(* IEC 61131-3 sources: AcpTrakStarwheel/TrkBufLib, 10 files *)

(* ---- Types.typ ---- *)
(*Buffer Base Type*)

TYPE
	tbAsyncShuttleBufferType : 	STRUCT  (*Asynchronous Buffer data*)
		ReadIdx : USINT; (*Starting index of the ring buffer*)
		WriteIdx : USINT; (*Ending index of the ring buffer*)
		Shuttles : ARRAY[0..tbMAX_BUF_IDX]OF McAxisType; (*Shuttles in the ring buffer*)
	END_STRUCT;
END_TYPE

(*Routed Move Velcity from Trigger Buffer*)

TYPE
	tbRtdMvVelTrgBufferParType : 	STRUCT  (*Parameters*)
		Position : LREAL; (*Position to send shuttle to*)
		RouteVelocity : REAL; (*Velocity of the shuttle before reaching the target position*)
		Velocity : REAL; (*Velocity of the shuttle after reaching the target position*)
		Acceleration : REAL; (*Acceleration of shuttle*)
		Deceleration : REAL; (*Deceleration of shuttle*)
		AdvancedParameters : McAcpTrakAdvRouteParType; (*Advanced move parameters*)
	END_STRUCT;
	tbRtdMvVelTrgBufferInternalType : 	STRUCT  (*Internal Data*)
		State : tbRtdTrgBufferStateEnum; (*State of execution*)
		TrgPointEnable : MC_BR_TrgPointEnable_AcpTrak; (*Enable process point*)
		TrgPointGetInfo : MC_BR_TrgPointGetInfo_AcpTrak; (*Get process point information*)
		RoutedMoveVel : MC_BR_RoutedMoveVel_AcpTrak; (*Move shuttle*)
		Status : DINT; (*Status*)
	END_STRUCT;
	tbRtdTrgBufferStateEnum :
		( (*State of execution for routed move from trigger*)
		tbRTD_TRG_BUF_STATE_IDLE, (*Idle state*)
		tbRTD_TRG_BUF_STATE_ENABLE_TRIG, (*Enable the process point*)
		tbRTD_TRG_BUF_STATE_GET_INFO, (*Get information from the start process point*)
		tbRTD_TRG_BUF_STATE_MOVE, (*Move shuttle*)
		tbRTD_TRG_BUF_STATE_RESET_FB, (*Reset function blocks*)
		tbRTD_TRG_BUF_STATE_NOT_BUSY, (*Wait for function blocks to report not busy*)
		tbRTD_TRG_BUF_STATE_ERROR (*An error occurred*)
		);
END_TYPE

(*Elastic Move Absolute from Position Buffer*)

TYPE
	tbElaMvAbsPosBufferParType : 	STRUCT  (*Parameters*)
		ArrivalPosition : LREAL; (*Position to wait for shuttles to arrive to*)
		DestinationPosition : LREAL; (*Position to send shuttles to*)
		DestinationVelocity : REAL; (*Velocity to move to destination*)
		DestinationAcceleration : REAL; (*Acceleration to move to destination*)
		DestinationDeceleration : REAL; (*Deceleration to move to destination*)
	END_STRUCT;
	tbElaMvAbsPosBufferInternalType : 	STRUCT  (*Internal Data*)
		State : tbElaPosBufferStateEnum; (*State of execution*)
		ShReadInfo : MC_BR_ShReadInfo_AcpTrak; (*Read shuttle info*)
		ElasticMoveAbs : MC_BR_ElasticMoveAbs_AcpTrak; (*Elastic move absolute*)
		Axis : McAxisType; (*Axis to control*)
		Status : DINT; (*Status*)
	END_STRUCT;
	tbElaPosBufferStateEnum :
		( (*State of execution*)
		tbELA_POS_BUF_STATE_IDLE, (*Idle state*)
		tbELA_POS_BUF_STATE_WAIT, (*Wait for a shuttle to be available*)
		tbELA_POS_BUF_STATE_POS, (*Wait for shuttle to reach the specified position on the sector*)
		tbELA_POS_BUF_STATE_MOVE, (*Move the shuttle to its position*)
		tbELA_POS_BUF_STATE_RESET_FB, (*Reset function blocks*)
		tbELA_POS_BUF_STATE_NOT_BUSY, (*Wait for function blocks to report not busy*)
		tbELA_POS_BUF_STATE_ERROR (*An error occurred*)
		);
END_TYPE

(* ---- BufferAddSh.st ---- *)
FUNCTION tbBufferAddSh

    IF ((Buffer.WriteIdx + 1) MOD (tbMAX_BUF_IDX + 1)) = Buffer.ReadIdx THEN
       tbBufferAddSh := tbERR_MAX_BUF_IDX;
    ELSE
        //Add the shuttle to the buffer
        brsmemcpy(ADR(Buffer.Shuttles[Buffer.WriteIdx]), ADR(Shuttle), SIZEOF(Buffer.Shuttles[Buffer.WriteIdx]));
        Buffer.WriteIdx := (Buffer.WriteIdx + 1) MOD (tbMAX_BUF_IDX + 1);
        tbBufferAddSh := ERR_OK;
    END_IF
    RETURN;

END_FUNCTION

(* ---- BufferGetFirst.st ---- *)
FUNCTION tbBufferGetFirst

    IF tbBufferShAvailable(ADR(Buffer)) THEN
        brsmemcpy(ADR(Shuttle), ADR(Buffer.Shuttles[Buffer.ReadIdx]), SIZEOF(Shuttle));
        tbBufferGetFirst := ERR_OK;
    ELSE
        tbBufferGetFirst := tbERR_NO_SH_IN_BUFFER;
    END_IF
    RETURN;

END_FUNCTION

(* ---- BufferRemoveFirst.st ---- *)
FUNCTION tbBufferRemoveFirst

    IF tbBufferShAvailable(ADR(Buffer)) THEN
        Buffer.ReadIdx := (Buffer.ReadIdx + 1) MOD (tbMAX_BUF_IDX + 1);
        tbBufferRemoveFirst := ERR_OK;
    ELSE
        tbBufferRemoveFirst := tbERR_NO_SH_IN_BUFFER;
    END_IF
    RETURN;

END_FUNCTION

(* ---- BufferShAvailable.st ---- *)
FUNCTION tbBufferShAvailable

    tbBufferShAvailable := Buffer.ReadIdx <> Buffer.WriteIdx;
    RETURN;

END_FUNCTION

(* ---- ShInBuffer.st ---- *)
FUNCTION tbShInBuffer

    i := Buffer.ReadIdx;
    WHILE i <> Buffer.WriteIdx DO
        IF brsmemcmp(ADR(Buffer.Shuttles[i]), ADR(Shuttle), SIZEOF(Buffer.Shuttles[i])) = 0 THEN
            tbShInBuffer := 1;
            RETURN;
        END_IF
        i := (i + 1) MOD (tbMAX_BUF_IDX + 1);
    END_WHILE
    tbShInBuffer := 0;
    RETURN;

END_FUNCTION

(* ---- ElasticMoveAbsPosBuffer.st ---- *)
FUNCTION_BLOCK tbElasticMoveAbsPosBuffer

    CASE Internal.State OF

        tbELA_POS_BUF_STATE_IDLE:

            IF Enable THEN
                Busy := 1;
                Active := 1;
                Internal.ShReadInfo.Axis := ADR(Internal.Axis);
                Internal.ElasticMoveAbs.Axis := ADR(Internal.Axis);
                Internal.State := tbELA_POS_BUF_STATE_WAIT;
            END_IF

        tbELA_POS_BUF_STATE_WAIT:

            IF NOT Enable THEN
                Active := 0;
                Internal.State := tbELA_POS_BUF_STATE_RESET_FB;
            ELSIF tbBufferShAvailable(ADR(BufferIn)) THEN
                //A shuttle is now available
                Internal.Status := tbBufferGetFirst(ADR(BufferIn), ADR(Internal.Axis));
                IF Internal.Status = ERR_OK THEN
                    //The shuttle axis was successfully obtained
                    IF tbShInBuffer(ADR(BufferOut), ADR(Internal.Axis)) THEN
                        //The shuttle already exists in the out buffer
                        Internal.Status := tbBufferRemoveFirst(ADR(BufferIn));
                        IF Internal.Status <> ERR_OK THEN
                            //An error occurred while removing the first shuttle from the buffer in
                            Active := 0;
                            Error := 1;
                            ErrorID := Internal.Status;
                            Internal.State := tbELA_POS_BUF_STATE_RESET_FB;
                        END_IF
                    ELSE
                        Internal.ShReadInfo.Enable := 1;
                        Internal.State := tbELA_POS_BUF_STATE_POS;
                    END_IF
                ELSE
                    //An error occurred while getting the shuttle axis
                    Active := 0;
                    Error := 1;
                    ErrorID := Internal.Status;
                    Internal.State := tbELA_POS_BUF_STATE_RESET_FB;
                END_IF
            END_IF

        tbELA_POS_BUF_STATE_POS:

            IF NOT Enable THEN
                Active := 0;
                Internal.State := tbELA_POS_BUF_STATE_RESET_FB;
            ELSIF Internal.ShReadInfo.Error THEN
                Active := 0;
                Error := 1;
                ErrorID := Internal.ShReadInfo.ErrorID;
                Internal.State := tbELA_POS_BUF_STATE_RESET_FB;

            ELSIF Internal.ShReadInfo.Valid AND
                  (Internal.ShReadInfo.ShuttleInfo.CurrentValues.SectorType <> mcACPTRAK_SEC_INTERNAL) AND
                  (Internal.ShReadInfo.ShuttleInfo.CurrentValues.Position >= Parameters.ArrivalPosition) THEN

                Internal.ShReadInfo.Enable := 0;
                Internal.ElasticMoveAbs.Position := Parameters.DestinationPosition;
                Internal.ElasticMoveAbs.Velocity := Parameters.DestinationVelocity;
                Internal.ElasticMoveAbs.Acceleration := Parameters.DestinationAcceleration;
                Internal.ElasticMoveAbs.Deceleration := Parameters.DestinationDeceleration;
                Internal.ElasticMoveAbs.Execute := 1;
                Internal.State := tbELA_POS_BUF_STATE_MOVE;

            END_IF

        tbELA_POS_BUF_STATE_MOVE:

            IF NOT Enable THEN
                Active := 0;
                Internal.State := tbELA_POS_BUF_STATE_RESET_FB;
            ELSIF Internal.ElasticMoveAbs.Error THEN
                Active := 0;
                Error := 1;
                ErrorID := Internal.ElasticMoveAbs.ErrorID;
                Internal.State := tbELA_POS_BUF_STATE_RESET_FB;
            ELSIF Internal.ElasticMoveAbs.Active OR Internal.ElasticMoveAbs.Done THEN
                Internal.ElasticMoveAbs.Execute := 0;
                Internal.Status := tbBufferRemoveFirst(ADR(BufferIn));
                IF Internal.Status = ERR_OK THEN
                    Internal.Status := tbBufferAddSh(ADR(BufferOut), ADR(Internal.Axis));
                    IF Internal.Status = ERR_OK THEN
                        Internal.State := tbELA_POS_BUF_STATE_WAIT;
                    ELSE
                        //An error occurred while adding the shuttle to the buffer out
                        Active := 0;
                        Error := 1;
                        ErrorID := Internal.Status;
                        Internal.State := tbELA_POS_BUF_STATE_RESET_FB;
                    END_IF
                ELSE
                    //An error occurred while removing the first shuttle from the buffer in
                    Active := 0;
                    Error := 1;
                    ErrorID := Internal.Status;
                    Internal.State := tbELA_POS_BUF_STATE_RESET_FB;
                END_IF
            END_IF

        tbELA_POS_BUF_STATE_RESET_FB:

            Internal.ShReadInfo.Enable := 0;
            Internal.ElasticMoveAbs.Execute := 0;
            IF Error THEN
                Internal.State := tbELA_POS_BUF_STATE_ERROR;
            ELSE
                Internal.State := tbELA_POS_BUF_STATE_NOT_BUSY;
            END_IF

        tbELA_POS_BUF_STATE_NOT_BUSY:

            IF NOT (Internal.ShReadInfo.Busy OR Internal.ElasticMoveAbs.Busy) THEN
                Busy := 0;
                Internal.State := tbELA_POS_BUF_STATE_IDLE;
            END_IF

        tbELA_POS_BUF_STATE_ERROR:

            IF NOT Enable THEN
                Error := 0;
                ErrorID := ERR_OK;
                Internal.State := tbELA_POS_BUF_STATE_NOT_BUSY;
            END_IF

    END_CASE

    Internal.ShReadInfo();
    Internal.ElasticMoveAbs();

END_FUNCTION_BLOCK

(* ---- RoutedMoveVelTrigBuffer.st ---- *)
FUNCTION_BLOCK tbRoutedMoveVelTrgBuffer

    CASE Internal.State OF

        tbRTD_TRG_BUF_STATE_IDLE:

            IF Enable THEN
                Busy := 1;
                Internal.TrgPointEnable.ProcessPoint := ADR(ProcessPoint);
                Internal.TrgPointEnable.Enable := 1;
                Internal.TrgPointGetInfo.ProcessPoint := ADR(ProcessPoint);
                Internal.RoutedMoveVel.Sector := ADR(Sector);
                Internal.RoutedMoveVel.Axis := ADR(Internal.TrgPointGetInfo.TrgPointInfo.Axis);
                Internal.State := tbRTD_TRG_BUF_STATE_ENABLE_TRIG;
            END_IF

        tbRTD_TRG_BUF_STATE_ENABLE_TRIG:

            IF Internal.TrgPointEnable.Valid THEN
                Active := 1;
            END_IF
            IF NOT Enable THEN
                Active := 0;
                Internal.State := tbRTD_TRG_BUF_STATE_RESET_FB;
            ELSIF Internal.TrgPointEnable.Error THEN
                Active := 0;
                Error := 1;
                ErrorID := Internal.TrgPointEnable.ErrorID;
                Internal.State := tbRTD_TRG_BUF_STATE_RESET_FB;
            ELSIF Internal.TrgPointEnable.Valid AND (Internal.TrgPointEnable.EventCount > 0) THEN
                Internal.TrgPointGetInfo.Execute := 1;
                Internal.State := tbRTD_TRG_BUF_STATE_GET_INFO;
            END_IF

        tbRTD_TRG_BUF_STATE_GET_INFO:

            IF NOT Enable THEN
                Active := 0;
                Internal.State := tbRTD_TRG_BUF_STATE_RESET_FB;
            ELSIF Internal.TrgPointGetInfo.Error THEN
                Active := 0;
                Error := 1;
                ErrorID := Internal.TrgPointGetInfo.ErrorID;
                Internal.State := tbRTD_TRG_BUF_STATE_RESET_FB;
            ELSIF Internal.TrgPointGetInfo.Done THEN
                IF tbShInBuffer(ADR(Buffer), ADR(Internal.TrgPointGetInfo.TrgPointInfo.Axis)) THEN
                    //The shuttle is already in the buffer
                    Internal.TrgPointGetInfo.Execute := 0;
                    Internal.State := tbRTD_TRG_BUF_STATE_ENABLE_TRIG;
                ELSE
                    //Continue adding the shuttle to the buffer
                    Internal.RoutedMoveVel.Position := Parameters.Position;
                    Internal.RoutedMoveVel.RouteVelocity := Parameters.RouteVelocity;
                    Internal.RoutedMoveVel.Velocity := Parameters.Velocity;
                    Internal.RoutedMoveVel.Acceleration := Parameters.Acceleration;
                    Internal.RoutedMoveVel.Deceleration := Parameters.Deceleration;
                    Internal.RoutedMoveVel.AdvancedParameters := Parameters.AdvancedParameters;
                    Internal.RoutedMoveVel.Execute := 1;
                    Internal.State := tbRTD_TRG_BUF_STATE_MOVE;
                END_IF
            END_IF

        tbRTD_TRG_BUF_STATE_MOVE:

            IF NOT Enable THEN
                Active := 0;
                Internal.State := tbRTD_TRG_BUF_STATE_RESET_FB;
            ELSIF Internal.RoutedMoveVel.Error THEN
                Active := 0;
                Error := 1;
                ErrorID := Internal.RoutedMoveVel.ErrorID;
                Internal.State := tbRTD_TRG_BUF_STATE_RESET_FB;
            ELSIF Internal.RoutedMoveVel.Active THEN
                Internal.TrgPointGetInfo.Execute := 0;
                Internal.RoutedMoveVel.Execute := 0;
                Internal.Status := tbBufferAddSh(ADR(Buffer), ADR(Internal.TrgPointGetInfo.TrgPointInfo.Axis));
                IF Internal.Status = ERR_OK THEN
                    //The shuttle was successfully added to the buffer
                    Internal.State := tbRTD_TRG_BUF_STATE_ENABLE_TRIG;
                ELSE
                    Active := 0;
                    Error := 1;
                    ErrorID := Internal.Status;
                    Internal.State := tbRTD_TRG_BUF_STATE_RESET_FB;
                END_IF
            END_IF

        tbRTD_TRG_BUF_STATE_RESET_FB:

            Internal.TrgPointEnable.Enable := 0;
            Internal.TrgPointGetInfo.Execute := 0;
            Internal.RoutedMoveVel.Execute := 0;
            IF Error THEN
                Internal.State := tbRTD_TRG_BUF_STATE_ERROR;
            ELSE
                Internal.State := tbRTD_TRG_BUF_STATE_NOT_BUSY;
            END_IF

        tbRTD_TRG_BUF_STATE_NOT_BUSY:

            IF NOT (Internal.TrgPointEnable.Busy OR Internal.TrgPointGetInfo.Busy OR Internal.RoutedMoveVel.Busy) THEN
                Busy := 0;
                Internal.State := tbRTD_TRG_BUF_STATE_IDLE;
            END_IF

        tbRTD_TRG_BUF_STATE_ERROR:

            IF NOT Enable THEN
                Error := 0;
                ErrorID := ERR_OK;
                Internal.State := tbRTD_TRG_BUF_STATE_NOT_BUSY;
            END_IF

    END_CASE

    Internal.TrgPointEnable();
    Internal.TrgPointGetInfo();
    Internal.RoutedMoveVel();

END_FUNCTION_BLOCK

(* ---- TrkBufLib.fun ---- *)
FUNCTION_BLOCK tbRoutedMoveVelTrgBuffer (*Monitor process point and perform routed move velocity before adding shuttle to buffer*)
	VAR_INPUT
		Sector : REFERENCE TO McSectorType; (*Target sector*)
		ProcessPoint : REFERENCE TO McProcessPointType; (*Process point to monitor*)
		Buffer : REFERENCE TO tbAsyncShuttleBufferType; (*Buffer*)
		Parameters : REFERENCE TO tbRtdMvVelTrgBufferParType; (*Parameters*)
		Enable : BOOL; (*Enable shuttle buffer*)
	END_VAR
	VAR_OUTPUT
		Busy : BOOL; (*The function block is busy and must continue to be called*)
		Active : BOOL; (*The buffer is active*)
		Error : BOOL; (*An error occurred*)
		ErrorID : DINT; (*ID of the error that occurred*)
	END_VAR
	VAR
		Internal : tbRtdMvVelTrgBufferInternalType; (*Internal Data*)
	END_VAR
END_FUNCTION_BLOCK

FUNCTION_BLOCK tbElasticMoveAbsPosBuffer (*Monitor a buffer for position to be exceeded and perform elastic move absolute before adding shuttle to buffer*)
	VAR_INPUT
		BufferIn : REFERENCE TO tbAsyncShuttleBufferType; (*Input buffer to monitor*)
		BufferOut : REFERENCE TO tbAsyncShuttleBufferType; (*Output buffer to write*)
		Parameters : REFERENCE TO tbElaMvAbsPosBufferParType; (*Parameters*)
		Enable : BOOL; (*Enable shuttle buffer*)
	END_VAR
	VAR_OUTPUT
		Busy : BOOL; (*The function block is busy and must continue to be called*)
		Active : BOOL; (*The buffer is active*)
		Error : BOOL; (*An error occurred*)
		ErrorID : DINT; (*ID of the error that occurred*)
	END_VAR
	VAR
		Internal : tbElaMvAbsPosBufferInternalType; (*Internal Data*)
	END_VAR
END_FUNCTION_BLOCK

FUNCTION tbBufferAddSh : DINT (*Add shuttle to the buffer*)
	VAR_INPUT
		Buffer : REFERENCE TO tbAsyncShuttleBufferType; (*Buffer to evaluate*)
		Shuttle : REFERENCE TO McAxisType; (*Shuttle to look for*)
	END_VAR
END_FUNCTION

FUNCTION tbBufferGetFirst : DINT (*Get the first shuttle entered in the buffer*)
	VAR_INPUT
		Buffer : REFERENCE TO tbAsyncShuttleBufferType; (*Buffer to evaluate*)
		Shuttle : REFERENCE TO McAxisType; (*First shuttle in the buffer*)
	END_VAR
END_FUNCTION

FUNCTION tbBufferRemoveFirst : DINT (*Remove the first shuttle entered in the buffer*)
	VAR_INPUT
		Buffer : REFERENCE TO tbAsyncShuttleBufferType; (*Buffer to modify*)
	END_VAR
END_FUNCTION

FUNCTION tbShInBuffer : BOOL (*Specified shuttle is in the buffer*)
	VAR_INPUT
		Buffer : REFERENCE TO tbAsyncShuttleBufferType; (*Buffer to evaluate*)
		Shuttle : REFERENCE TO McAxisType; (*Shuttle to look for*)
	END_VAR
	VAR
		i : USINT; (*Index*)
	END_VAR
END_FUNCTION

FUNCTION tbBufferShAvailable : BOOL (*A shuttle is available in the buffer*)
	VAR_INPUT
		Buffer : REFERENCE TO tbAsyncShuttleBufferType; (*Buffer to evaluate*)
	END_VAR
END_FUNCTION

(* ---- Constants.var ---- *)
(*Values*)
VAR CONSTANT
	tbMAX_BUF_IDX : USINT := 64; (*Maximum shuttle index in the buffer*)
END_VAR
(*Errors*)
VAR CONSTANT
	tbERR_MAX_BUF_IDX : DINT := -5500; (*Index of shuttle in buffer exceeds limit*)
	tbERR_NO_SH_IN_BUFFER : DINT := -5501; (*No shuttles are in the buffer*)
END_VAR
